FUNCTION_BLOCK FB_PieceBase EXTENDS FB_Object
VAR_INPUT
END_VAR
VAR_OUTPUT
	bUsingPiece			: BOOL;	
END_VAR
VAR
	pParentObject		: POINTER TO FB_Object;
	stDimension			: ST_3DDimension;
	rSlotDiameter		: REAL;
	stOffset			: ST_3DPoint;	//Offset
	rZOverlapTool		: REAL;
	rZOverlapSlot		: REAL;
	rMeasureDistance	: REAL;
	rDockOffset			: REAL;
	nCurrentPropIndex	: USINT;
	nSpecPropIndex		: USINT;			//erster Index für Specialproperties
	bIgnoreOffset		: BOOL;
END_VAR

METHOD M_UpdateParent
VAR_INPUT
END_VAR
IF pObjCollectNode > 0 AND_THEN pObjCollectNode^.pOwnerColl > 0 THEN
	pParentObject := pObjCollectNode^.pOwnerColl^.pOwnerNode^.P_pObject;
ELSE
	pParentObject := 0;
END_IF

IF pParentObject > 0 THEN
	pParentSlot := pParentObject^.M_GetSlotFromChild(THIS);
ELSE
	pParentSlot := 0;
END_IF
END_METHOD

METHOD M_GetPropCheckSum : UINT
VAR_INPUT
END_VAR

VAR
	stData 		: ST_CmdData;
END_VAR
M_GetAllProps(stData);
wChecksum := F_DATA_TO_CRC16_CCITT(ADR(stData.n32Data[0]),nNoOfProps * 4,16#FFFF);
M_GetPropCheckSum := wChecksum;
END_METHOD

PROPERTY P_stDimension : ST_3DDimension
GET
P_stDimension := stDimension;
END_GET
END_PROPERTY

PROPERTY P_rDockOffset : REAL
GET
P_rDockOffset := rDockOffset;
END_GET
END_PROPERTY

{attribute 'object_name' := 'M_CheckProps'}
METHOD M_CheckProps : ERRORID
END_METHOD

PROPERTY P_rZOverlapSlot : REAL
GET
P_rZOverlapSlot := rZOverlapSlot;
END_GET
END_PROPERTY

PROPERTY P_pLatestChild : POINTER TO FB_PieceBase
GET
P_pLatestChild := THIS;
END_GET
END_PROPERTY

PROPERTY P_rZOverlapTool : REAL
GET
P_rZOverlapTool := rZOverlapTool;
END_GET
END_PROPERTY

PROPERTY P_stOffset : ST_3DPoint
GET
P_stOffset := stOffset;
END_GET
SET
stOffset := P_stOffset;
END_SET
END_PROPERTY

{attribute 'object_name' := 'M_ClearAllProps'}
METHOD M_ClearAllProps

VAR_INPUT
	bIgnoreParent : BOOL; //Es wird das gesamte OD gelöscht. -> Zeiger auf Parent nicht mehr gültig!
END_VAR
IF NOT bIgnoreParent THEN
	IF pParentSlot > 0 THEN
		pParentSlot^.P_pChild := 0;
	END_IF	
END_IF
nObjectID := 0;
pParentObject := 0;
pParentSlot := 0;
pObjCollectNode := 0;
END_METHOD

METHOD M_GetRelPosTopCenter : ST_3DPoint
VAR_INPUT
END_VAR
VAR
	stPosTemp : ST_3DPoint;
	pPieceSlot : POINTER TO FB_PieceSlot;
END_VAR
IF pParentObject > 0 THEN
	IF pParentObject^.M_bIsGroup(E_ObjectGroup.OBJECTGROUP_Target) THEN
		IF pParentSlot > 0 THEN
			pPieceSlot := pParentSlot;
			stPosTemp := pPieceSlot^.P_stRelPos;
			//Wenn OverlapSlot > SlotTiefe, dann sitzt Piece auf dem Grund des Slots auf
			IF rZOverlapSlot > pPieceSlot^.rDepth THEN
				stPosTemp.Z := stPosTemp.Z - pPieceSlot^.rDepth + stDimension.Height;
			ELSE
				stPosTemp.Z := stPosTemp.Z - rZOverlapSlot + stDimension.Height;
			END_IF
			IF bIgnoreOffset THEN
				M_GetRelPosTopCenter := stPosTemp;
			ELSE
				M_GetRelPosTopCenter := F_Add3DPoints(stPosTemp,stOffset);	
			END_IF
		END_IF
	END_IF
END_IF
END_METHOD

{attribute 'object_name' := 'M_SetSingleProp'}
METHOD M_SetSingleProp : ERRORID
VAR_INPUT
	refCmdData	: REFERENCE TO ST_CmdData;
END_VAR
CASE refCmdData.aHeader[1] OF
	0,1:
		M_SetSingleProp := E_ErrorIdCmd.ERRORID_InvalidProperty;
	2:	stDimension.Width := DINT_TO_REAL(refCmdData.n32Data[0]);
	3:	stDimension.Depth := DINT_TO_REAL(refCmdData.n32Data[0]);
	4:	stDimension.Height := DINT_TO_REAL(refCmdData.n32Data[0]);
	5:	rSlotDiameter := DINT_TO_REAL(refCmdData.n32Data[0]);
	6:	rZOverlapTool := DINT_TO_REAL(refCmdData.n32Data[0]);
	7:	rZOverlapSlot := DINT_TO_REAL(refCmdData.n32Data[0]);
	8:	stOffset.X := DINT_TO_REAL(refCmdData.n32Data[0]);
	9:	stOffset.Y := DINT_TO_REAL(refCmdData.n32Data[0]);
	10:	stOffset.Z := DINT_TO_REAL(refCmdData.n32Data[0]);
	11: rMeasureDistance := DINT_TO_REAL(refCmdData.n32Data[0]);
	12:	rDockOffset := DINT_TO_REAL(refCmdData.n32Data[0]);
END_CASE
END_METHOD

METHOD M_ClearOffset
VAR_INPUT
END_VAR
stOffset.X := 0.0;
stOffset.Y := 0.0;
stOffset.Z := 0.0;
END_METHOD

PROPERTY P_rMeasureDistance : REAL
GET
P_rMeasureDistance := rMeasureDistance;
END_GET
END_PROPERTY

{attribute 'object_name' := 'M_GetAllProps'}
METHOD M_GetAllProps : ERRORID
VAR_INPUT
	refCmdData	: REFERENCE TO ST_CmdData;
END_VAR
refCmdData.aHeader[0] := nObjectID;
refCmdData.aHeader[1] := eObjectType;
refCmdData.aHeader[2] := 0;

IF pParentObject > 0 THEN
	refCmdData.n32Data[0] := pParentObject^.P_nObjectID;
ELSE
	refCmdData.n32Data[0] := 0;
END_IF

IF pParentSlot > 0 THEN
	refCmdData.n32Data[1] := pParentSlot^.nNr;
ELSE
	refCmdData.n32Data[1] := 0;
END_IF

//Dimensionen lesen
refCmdData.n32Data[2] := REAL_TO_DINT(stDimension.Width);
refCmdData.n32Data[3] := REAL_TO_DINT(stDimension.Depth);
refCmdData.n32Data[4] := REAL_TO_DINT(stDimension.Height);
refCmdData.n32Data[5] := REAL_TO_DINT(rSlotDiameter);
refCmdData.n32Data[6] := REAL_TO_DINT(rZOverlapTool);
refCmdData.n32Data[7] := REAL_TO_DINT(rZOverlapSlot);
refCmdData.n32Data[8] := REAL_TO_DINT(stOffset.X);
refCmdData.n32Data[9] := REAL_TO_DINT(stOffset.Y);
refCmdData.n32Data[10] := REAL_TO_DINT(stOffset.Z);
refCmdData.n32Data[11] := REAL_TO_DINT(rMeasureDistance);
refCmdData.n32Data[12] := REAL_TO_DINT(rDockOffset);
nCurrentPropIndex := 12;
END_METHOD

METHOD M_AddChild : ERRORID
VAR_INPUT
	pObject	: POINTER TO FB_Object;
	nSlotNr	: UINT;
	nIndex 	: INT;
END_VAR
//Pieces könnnen keine Childs aufnehmen
M_AddChild := E_ErrorIdObjMgmt.ERRORID_ObjectCanNotTakeChilds;
END_METHOD

{attribute 'object_name' := 'M_SetAllProps'}
METHOD M_SetAllProps : ERRORID
VAR_INPUT
	refCmdData	: REFERENCE TO ST_CmdData;
END_VAR
IF fbObjectDirectory.M_GetObjPointer(DINT_TO_UINT(refCmdData.n32Data[0])) = 0 THEN
	M_SetAllProps := E_ErrorIdObjMgmt.ERRORID_InvalidParentObject;
	RETURN;
END_IF

//ParentSlot unterschiedlich?

(*IF pParentSlot = 0 THEN
	M_SetAllProps := M_SetParent(aI_Object[refCmdData.n32Data[0]],DINT_TO_UINT(refCmdData.n32Data[1]));
ELSE
	IF pParentSlot^.P_nNr <> DINT_TO_UINT(refCmdData.n32Data[1]) THEN
		M_SetAllProps := M_SetParent(aI_Object[refCmdData.n32Data[0]],DINT_TO_UINT(refCmdData.n32Data[1]));
	END_IF
END_IF

IF M_SetAllProps > 0 THEN
	RETURN;
END_IF*)

//Dimensionen setzen
stDimension.Width := DINT_TO_REAL(refCmdData.n32Data[2]);
stDimension.Depth := DINT_TO_REAL(refCmdData.n32Data[3]);
stDimension.Height := DINT_TO_REAL(refCmdData.n32Data[4]);
rSlotDiameter := DINT_TO_REAL(refCmdData.n32Data[5]);
rZOverlapTool := DINT_TO_REAL(refCmdData.n32Data[6]);
rZOverlapSlot := DINT_TO_REAL(refCmdData.n32Data[7]);
stOffset.X := DINT_TO_REAL(refCmdData.n32Data[8]);
stOffset.Y := DINT_TO_REAL(refCmdData.n32Data[9]);
stOffset.Z := DINT_TO_REAL(refCmdData.n32Data[10]);
rMeasureDistance := DINT_TO_REAL(refCmdData.n32Data[11]);
rDockOffset := DINT_TO_REAL(refCmdData.n32Data[12]);
nCurrentPropIndex := 12;
nNoOfProps := nCurrentPropIndex + 1;
END_METHOD

PROPERTY P_nCntSlots : UINT
GET
END_GET
END_PROPERTY

PROPERTY P_bIgnoreOffset : BOOL
SET
bIgnoreOffset := P_bIgnoreOffset;
END_SET
GET
P_bIgnoreOffset := bIgnoreOffset;
END_GET
END_PROPERTY

END_FUNCTION_BLOCK

(* stored: Version 1.1.0.1
   POU FB_PieceBase: Id {63b07fb9-5ab1-4920-9bfc-a43e0b6ab977}, SpecialFunc None
   Method M_UpdateParent: Id {12272a62-205a-4dc2-ab64-81302efaa155}
   Method M_GetPropCheckSum: Id {18633363-fac8-4800-9b10-f9ba3b401402}
   Property P_stDimension: Id {38cfc3fb-8369-4149-a7c6-1e896656ace3}
   Get Get: Id {583f7b0b-c4be-47cf-978b-40ce2de136c8}
   Property P_rDockOffset: Id {51558094-4c39-411f-879f-5d616be5f64f}
   Get Get: Id {f60d6112-2c55-486f-8f1e-da6ce27be520}
   Method M_CheckProps: Id {55fc7aaa-cef2-4c3c-8779-ab7d9e3b0219}
   Property P_rZOverlapSlot: Id {567ff299-7005-4f6d-a9e8-9c08dff96786}
   Get Get: Id {9407881e-c1e3-4504-8457-e2ec5cb609f1}
   Property P_pLatestChild: Id {599afd22-374e-473d-8028-cebee4c6bece}
   Get Get: Id {c8f06d56-fe69-4d12-9409-8169bbd8a26b}
   Property P_rZOverlapTool: Id {5e5f6762-008e-42af-8d8d-704a3888c52c}
   Get Get: Id {2fcd534d-4388-454b-8be3-60a5ae57e755}
   Property P_stOffset: Id {604faea7-ad93-4a8b-aef7-91a75165f3a7}
   Get Get: Id {328cfb13-c842-4ea7-948d-177437d03342}
   Set Set: Id {50a76d6a-1900-4314-80fa-1453c6d08102}
   Method M_ClearAllProps: Id {7719d9df-58e4-46b7-b1d8-5dfd54045015}
   Method M_GetRelPosTopCenter: Id {895bb838-4287-4255-85e0-880c3d6350cd}
   Method M_SetSingleProp: Id {8b42104b-9230-4634-bf32-5bb53ab65987}
   Method M_ClearOffset: Id {8ce0672d-aa64-4446-b80a-5f086ed20313}
   Property P_rMeasureDistance: Id {9bae66cb-d201-4dcc-8eb2-a70f9ca72cb0}
   Get Get: Id {62c0c84e-0df8-4c92-befd-d44a6bd21024}
   Method M_GetAllProps: Id {b457f268-2efd-4fe4-9c95-d0bca3e91460}
   Method M_AddChild: Id {bcc24b54-37c5-4672-ac4e-4def77d6218c}
   Method M_SetAllProps: Id {c95aee18-be78-4b3d-b6ed-71f97931af31}
   Property P_nCntSlots: Id {d7709e70-a5a5-43ae-94bf-2392db318ccf}
   Get Get: Id {59ce1092-2756-4af6-bc8d-f8ce2ec685e0}
   Property P_bIgnoreOffset: Id {e2645d6a-d2f5-4d76-a453-6a748247d97d}
   Set Set: Id {a745faca-8da2-4bd8-973c-ee532bfc2459}
   Get Get: Id {b505df4d-b201-4c10-bcff-6c2ca5f75af7} *)
